FUNCTION_BLOCK SAVING_PICKLE
  {SET_ATTRIBUTE(OpcUa, SERVICE)}
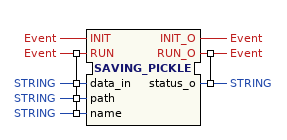
  EVENT_INPUT
    INIT;
    RUN WITH data_in, path, name; {SET_ATTRIBUTE(OpcUa, Method)}
  END_EVENT
  EVENT_OUTPUT
    INIT_O;
    RUN_O WITH status_o;
  END_EVENT
  VAR_INPUT
    data_in : STRING; {SET_ATTRIBUTE(OpcUa, Variable.RUN)}
    path : STRING; {SET_ATTRIBUTE(OpcUa, Variable.RUN)}
    name : STRING; {SET_ATTRIBUTE(OpcUa, Variable.RUN)}
  END_VAR
  VAR_OUTPUT
    status_o : STRING; {SET_ATTRIBUTE(OpcUa, Variable.RUN)}
  END_VAR
END_FUNCTION_BLOCK
